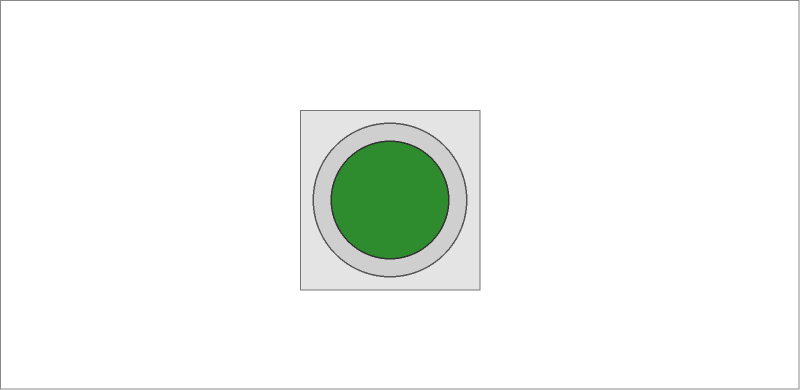
VISUALIZATION VisuDigitalOutControl  // 800x390
VAR_IN_OUT
	fbManualControler	: FB_ManualController ;
END_VAR
    PushSwitch (300,110 180x180), variable: fbManualControler.pDevDigitalOut^.bCmdOn, behaviour: TOGGLE, style: Switch-PushSwitch-Green
END_VISUALIZATION

(* stored: Version 1.1.0.1, ProductVersion 3.1.4024.9
   Visu VisuDigitalOutControl: Id {95b8514e-4195-4ad3-a984-a4f77012140d} *)
